(* IEC 61131-3 sources: com.logicals.lc3.webinar/usRTS_RPMControl_iSOC/src_FB_LIB_SAFE/Convert/UINT, 5 files *)

(* ---- wTRUNC_UINT_TO_USINT.iecst ---- *)
NAMESPACE logicals.web.standard
NAMESPACE convert

/*
 * Function block wrapper for IEC 61131-3 TO_USINT<br>
 * IN =  input value (UINT)<br>
 * OUT = IN (USINT)<br>
 */
FUNCTION_BLOCK wTRUNC_UINT_TO_USINT
	{ vNameAlignment:="center"; altName:="TRUNC_UINT_TO_USINT"; bgColor:="Plum"; width:=180; hideIONames; }
	VAR_INPUT
		IN : UINT;
	END_VAR
	VAR_OUTPUT
		OUT: USINT;
	END_VAR

	OUT := TO_USINT(IN:=IN, ENO=>ENO);
END_FUNCTION_BLOCK

END_NAMESPACE
END_NAMESPACE

(* ---- wUINT_TO_DINT.iecst ---- *)
NAMESPACE logicals.web.standard
NAMESPACE convert

/*
 * Function block wrapper for IEC 61131-3 TO_DINT<br>
 * IN =  input value (UINT)<br>
 * OUT = IN (DINT)<br>
 */
FUNCTION_BLOCK wUINT_TO_DINT
	{ vNameAlignment:="center"; altName:="UINT_TO_DINT"; bgColor:="LightPink"; width:=140; hideIONames; }
	VAR_INPUT
		IN : UINT;
	END_VAR
	VAR_OUTPUT
		OUT: DINT;
	END_VAR

	OUT := TO_DINT(IN:=IN, ENO=>ENO);
END_FUNCTION_BLOCK

END_NAMESPACE
END_NAMESPACE

(* ---- wUINT_TO_UDINT.iecst ---- *)
NAMESPACE logicals.web.standard
NAMESPACE convert

/*
 * Function block wrapper for IEC 61131-3 TO_UDINT<br>
 * IN =  input value (UINT)<br>
 * OUT = IN (UDINT)<br>
 */
FUNCTION_BLOCK wUINT_TO_UDINT
	{ vNameAlignment:="center"; altName:="UINT_TO_UDINT"; bgColor:="Plum"; width:=140; hideIONames; }
	VAR_INPUT
		IN : UINT;
	END_VAR
	VAR_OUTPUT
		OUT: UDINT;
	END_VAR

	OUT := TO_UDINT(IN:=IN, ENO=>ENO);
END_FUNCTION_BLOCK

END_NAMESPACE
END_NAMESPACE

(* ---- wUINT_TO_ULINT.iecst ---- *)
NAMESPACE logicals.web.standard
NAMESPACE convert

/*
 * Function block wrapper for IEC 61131-3 TO_ULINT<br>
 * IN =  input value (UINT)<br>
 * OUT = IN (ULINT)<br>
 */
FUNCTION_BLOCK wUINT_TO_ULINT
	{ vNameAlignment:="center"; altName:="UINT_TO_ULINT"; bgColor:="Plum"; width:=140; hideIONames; }
	VAR_INPUT
		IN : UINT;
	END_VAR
	VAR_OUTPUT
		OUT: ULINT;
	END_VAR

	OUT := TO_ULINT(IN:=IN, ENO=>ENO);
END_FUNCTION_BLOCK

END_NAMESPACE
END_NAMESPACE

(* ---- wUINT_TO_WORD.iecst ---- *)
NAMESPACE logicals.web.standard
NAMESPACE convert

/*
 * Function block wrapper for IEC 61131-3 TO_WORD<br>
 * IN =  input value (UINT)<br>
 * OUT = IN (WORD)<br>
 */
FUNCTION_BLOCK wUINT_TO_WORD
	{ vNameAlignment:="center"; altName:="UINT_TO_WORD"; bgColor:="DodgerBlue"; width:=140; hideIONames; }
	VAR_INPUT
		IN : UINT;
	END_VAR
	VAR_OUTPUT
		OUT: WORD;
	END_VAR

	OUT := TO_WORD(IN:=IN, ENO=>ENO);
END_FUNCTION_BLOCK

END_NAMESPACE
END_NAMESPACE
